ABB RAPID module: Module1.mod

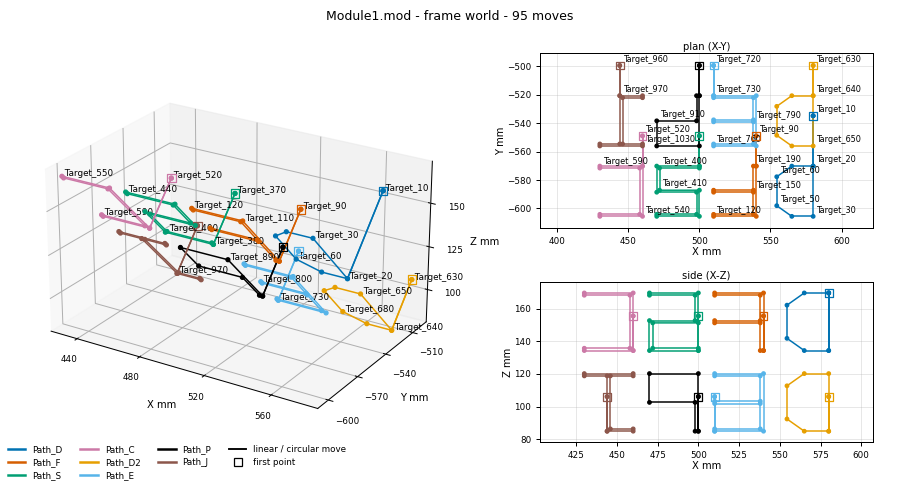
[picture p0: tool path of Module1.mod in frame world, 95 of 99 moves have a stored position in this frame; points joined in program order, loops and branches not executed]
MODULE Module1




    PERS tooldata PortaMarcadorTCP:=[TRUE,[[0,0,152],[1,0,0,0]],[0.15,[0,0,65],[1,0,0,0],0,0,0]];
    TASK PERS wobjdata Tablero_Inclinado:=[FALSE,TRUE,"",[[600,-619.706,183.848],[0,0,0.923879533,-0.382683432]],[[0,0,0],[1,0,0,0]]];
    CONST robtarget Target_10:=[[20,70,-50],[1,0,0,0],[-1,-1,0,0],[9E+09,9E+09,9E+09,9E+09,9E+09,9E+09]];
    CONST robtarget Target_20:=[[20,70.000430916,-0.000095827],[1,0,0,0],[-1,-1,0,0],[9E+09,9E+09,9E+09,9E+09,9E+09,9E+09]];
    CONST robtarget Target_30:=[[20,20.000430915,-0.00009588],[1,0,0,0],[-1,-1,0,0],[9E+09,9E+09,9E+09,9E+09,9E+09,9E+09]];
    CONST robtarget Target_40:=[[35,20.000430915,-0.00009588],[1,0,0,0],[-1,-1,0,0],[9E+09,9E+09,9E+09,9E+09,9E+09,9E+09]];
    CONST robtarget Target_50:=[[45.606601718,30.607032633,-0.000095869],[1,0.000000001,0,0],[-1,-1,0,0],[9E+09,9E+09,9E+09,9E+09,9E+09,9E+09]];
    CONST robtarget Target_60:=[[45.606601718,59.393829198,-0.000095838],[1,0,0,0],[-1,-1,0,0],[9E+09,9E+09,9E+09,9E+09,9E+09,9E+09]];
    CONST robtarget Target_70:=[[35,70.000430916,-0.000095827],[1,0.000000001,0,0],[-1,-1,0,0],[9E+09,9E+09,9E+09,9E+09,9E+09,9E+09]];
    CONST robtarget Target_80:=[[20,70.000430916,-0.000095827],[1,0,0,0],[0,0,0,0],[9E+09,9E+09,9E+09,9E+09,9E+09,9E+09]];
    CONST robtarget Target_10_2:=[[20,70,-50],[1,0,0,0],[-1,-1,0,0],[9E+09,9E+09,9E+09,9E+09,9E+09,9E+09]];
    CONST robtarget Target_90:=[[60,70.000430947,-30.000095827],[1,0,0,0],[0,0,0,0],[9E+09,9E+09,9E+09,9E+09,9E+09,9E+09]];
    CONST robtarget Target_100:=[[60,70.000430916,-0.000095827],[1,0,0,0],[-1,-1,0,0],[9E+09,9E+09,9E+09,9E+09,9E+09,9E+09]];
    CONST robtarget Target_110:=[[60,20.000430915,-0.00009588],[1,0,0,0],[-1,-1,0,0],[9E+09,9E+09,9E+09,9E+09,9E+09,9E+09]];
    CONST robtarget Target_120:=[[90,20.000430915,-0.00009588],[1,0,0,0],[-1,-2,0,0],[9E+09,9E+09,9E+09,9E+09,9E+09,9E+09]];
    CONST robtarget Target_130:=[[90,22.000430916,-0.000095877],[1,0,0,0],[-1,-2,0,0],[9E+09,9E+09,9E+09,9E+09,9E+09,9E+09]];
    CONST robtarget Target_140:=[[62,22.000430916,-0.000095877],[1,0,0,0],[-1,-1,0,0],[9E+09,9E+09,9E+09,9E+09,9E+09,9E+09]];
    CONST robtarget Target_150:=[[62,44.000430916,-0.000095854],[1,0,0,0],[-1,-1,0,0],[9E+09,9E+09,9E+09,9E+09,9E+09,9E+09]];
    CONST robtarget Target_160:=[[90,44.000430539,-0.000095855],[1,0,0,0],[-1,-2,0,0],[9E+09,9E+09,9E+09,9E+09,9E+09,9E+09]];
    CONST robtarget Target_170:=[[90,46.000430916,-0.000095852],[1,0,0,0],[-1,-2,0,0],[9E+09,9E+09,9E+09,9E+09,9E+09,9E+09]];
    CONST robtarget Target_180:=[[62,46.000430916,-0.000095852],[1,0,0,0],[-1,-1,0,0],[9E+09,9E+09,9E+09,9E+09,9E+09,9E+09]];
    CONST robtarget Target_190:=[[62,70.000430916,-0.000095827],[1,0,0,0],[-1,-2,0,0],[9E+09,9E+09,9E+09,9E+09,9E+09,9E+09]];
    CONST robtarget Target_200:=[[60,70.000430916,-0.000095827],[1,0,0,0],[-1,-1,0,0],[9E+09,9E+09,9E+09,9E+09,9E+09,9E+09]];
    CONST robtarget Target_210:=[[60,70.000430947,-30.000095827],[1,0,0,0],[-1,-1,0,0],[9E+09,9E+09,9E+09,9E+09,9E+09,9E+09]];
    CONST robtarget Target_370:=[[100,70.000430703,-30.000095827],[1,0,0,0],[-1,-2,0,0],[9E+09,9E+09,9E+09,9E+09,9E+09,9E+09]];
    CONST robtarget Target_380:=[[100,70.00043067,-0.000095827],[1,0,0,0],[-1,-2,0,0],[9E+09,9E+09,9E+09,9E+09,9E+09,9E+09]];
    CONST robtarget Target_390:=[[100,68.000430671,-0.000095829],[1,0,0,0],[-1,-2,0,0],[9E+09,9E+09,9E+09,9E+09,9E+09,9E+09]];
    CONST robtarget Target_400:=[[128,68.000430671,-0.000095829],[1,0,0,0],[-1,-2,0,0],[9E+09,9E+09,9E+09,9E+09,9E+09,9E+09]];
    CONST robtarget Target_410:=[[127.999999808,46.000430671,-0.000095852],[1,0,0,0],[-1,-2,0,0],[9E+09,9E+09,9E+09,9E+09,9E+09,9E+09]];
    CONST robtarget Target_420:=[[100,45.997147496,-0.000095852],[1,0.000000001,0,0],[-1,-2,0,0],[9E+09,9E+09,9E+09,9E+09,9E+09,9E+09]];
    CONST robtarget Target_430:=[[100,20.000430915,-0.00009588],[1,0,0,0],[-1,-2,0,0],[9E+09,9E+09,9E+09,9E+09,9E+09,9E+09]];
    CONST robtarget Target_440:=[[130,20.000430915,-0.00009588],[1,0,0,0],[-1,-2,0,0],[9E+09,9E+09,9E+09,9E+09,9E+09,9E+09]];
    CONST robtarget Target_450:=[[130,22.000430916,-0.000095877],[1,0,0,0],[-1,-2,0,0],[9E+09,9E+09,9E+09,9E+09,9E+09,9E+09]];
    CONST robtarget Target_460:=[[102,22.000430916,-0.000095877],[1,0,0,0],[-1,-2,0,0],[9E+09,9E+09,9E+09,9E+09,9E+09,9E+09]];
    CONST robtarget Target_470:=[[102,44.000430916,-0.000095854],[1,0,0,0],[-1,-2,0,0],[9E+09,9E+09,9E+09,9E+09,9E+09,9E+09]];
    CONST robtarget Target_480:=[[130,44.00043067,-0.000095855],[1,0,0,0],[-1,-2,0,0],[9E+09,9E+09,9E+09,9E+09,9E+09,9E+09]];
    CONST robtarget Target_490:=[[130,70.00043067,-0.000095827],[1,0,0,0],[-1,-2,0,0],[9E+09,9E+09,9E+09,9E+09,9E+09,9E+09]];
    CONST robtarget Target_500:=[[100,70.00043067,-0.000095827],[1,0,0,0],[-1,-2,0,0],[9E+09,9E+09,9E+09,9E+09,9E+09,9E+09]];
    CONST robtarget Target_510:=[[100,70.000430703,-30.000095827],[1,0,0,0],[-1,-2,0,0],[9E+09,9E+09,9E+09,9E+09,9E+09,9E+09]];
    CONST robtarget Target_520:=[[140,70.000430947,-30.000095827],[1,0,0,0],[-1,-2,0,0],[9E+09,9E+09,9E+09,9E+09,9E+09,9E+09]];
    CONST robtarget Target_530:=[[140,70.000430916,-0.000095827],[1,0,0,0],[-1,-2,0,0],[9E+09,9E+09,9E+09,9E+09,9E+09,9E+09]];
    CONST robtarget Target_540:=[[140,20.000430915,-0.00009588],[1,0,0,0],[-1,-2,0,0],[9E+09,9E+09,9E+09,9E+09,9E+09,9E+09]];
    CONST robtarget Target_550:=[[170,20.000430915,-0.00009588],[1,0,0,0],[-1,-2,0,0],[9E+09,9E+09,9E+09,9E+09,9E+09,9E+09]];
    CONST robtarget Target_560:=[[170,22.000431324,-0.000095877],[1,0,0,0],[-1,-2,0,0],[9E+09,9E+09,9E+09,9E+09,9E+09,9E+09]];
    CONST robtarget Target_570:=[[142,22.000430916,-0.000095877],[1,0,0,0],[-1,-2,0,0],[9E+09,9E+09,9E+09,9E+09,9E+09,9E+09]];
    CONST robtarget Target_580:=[[142,68.000430916,-0.000095829],[1,0,0,0],[-1,-2,0,0],[9E+09,9E+09,9E+09,9E+09,9E+09,9E+09]];
    CONST robtarget Target_590:=[[170,68.000430916,-0.000095829],[1,0,0,0],[-1,-2,0,0],[9E+09,9E+09,9E+09,9E+09,9E+09,9E+09]];
    CONST robtarget Target_600:=[[170,70.000430916,-0.000095827],[1,0,0,0],[-1,-2,0,0],[9E+09,9E+09,9E+09,9E+09,9E+09,9E+09]];
    CONST robtarget Target_610:=[[140,70.000430916,-0.000095827],[1,0,0,0],[-1,-2,0,0],[9E+09,9E+09,9E+09,9E+09,9E+09,9E+09]];
    CONST robtarget Target_620:=[[140,70.000430947,-30.000095827],[1,0,0,0],[-1,-2,0,0],[9E+09,9E+09,9E+09,9E+09,9E+09,9E+09]];
    CONST jointtarget PosicionInicial:=[[0,0,0,0,0,0],[9E+09,9E+09,9E+09,9E+09,9E+09,9E+09]];
    CONST jointtarget Intermedio:=[[0,30,0,0,0,0],[9E+09,9E+09,9E+09,9E+09,9E+09,9E+09]];
    CONST robtarget Target_630:=[[20,140.000430947,-30.000095754],[1,0,0,0],[0,0,0,0],[9E+09,9E+09,9E+09,9E+09,9E+09,9E+09]];
    CONST robtarget Target_640:=[[20,140.000430916,-0.000095753],[1,0,0,0],[0,0,0,0],[9E+09,9E+09,9E+09,9E+09,9E+09,9E+09]];
    CONST robtarget Target_650:=[[20,90.000430915,-0.000095806],[1,0,0,0],[0,0,0,0],[9E+09,9E+09,9E+09,9E+09,9E+09,9E+09]];
    CONST robtarget Target_660:=[[35,90.000430915,-0.000095806],[1,0,0,0],[0,0,0,0],[9E+09,9E+09,9E+09,9E+09,9E+09,9E+09]];
    CONST robtarget Target_670:=[[45.606601718,100.607032633,-0.000095795],[1,0.000000001,0,0],[0,0,0,0],[9E+09,9E+09,9E+09,9E+09,9E+09,9E+09]];
    CONST robtarget Target_680:=[[45.606601718,129.393829198,-0.000095764],[1,0,0,0],[0,0,0,0],[9E+09,9E+09,9E+09,9E+09,9E+09,9E+09]];
    CONST robtarget Target_690:=[[35,140.000430916,-0.000095753],[1,0.000000001,0,0],[0,0,0,0],[9E+09,9E+09,9E+09,9E+09,9E+09,9E+09]];
    CONST robtarget Target_700:=[[20,140.000430916,-0.000095753],[1,0,0,0],[0,0,0,0],[9E+09,9E+09,9E+09,9E+09,9E+09,9E+09]];
    CONST robtarget Target_710:=[[20,140.000430947,-30.000095754],[1,0,0,0],[0,0,0,0],[9E+09,9E+09,9E+09,9E+09,9E+09,9E+09]];
    CONST robtarget Target_720:=[[90,140.000430947,-30.000095754],[1,0,0,0],[0,0,0,0],[9E+09,9E+09,9E+09,9E+09,9E+09,9E+09]];
    CONST robtarget Target_730:=[[90,140.000430916,-0.000095753],[1,0,0,0],[0,0,0,0],[9E+09,9E+09,9E+09,9E+09,9E+09,9E+09]];
    CONST robtarget Target_740:=[[60,140.000430916,-0.000095753],[1,0,0,0],[0,0,0,0],[9E+09,9E+09,9E+09,9E+09,9E+09,9E+09]];
    CONST robtarget Target_750:=[[60,90.000430915,-0.000095806],[1,0,0,0],[0,0,0,0],[9E+09,9E+09,9E+09,9E+09,9E+09,9E+09]];
    CONST robtarget Target_760:=[[90,90.000430915,-0.000095806],[1,0,0,0],[0,0,0,0],[9E+09,9E+09,9E+09,9E+09,9E+09,9E+09]];
    CONST robtarget Target_770:=[[90,92.000430916,-0.000095803],[1,0,0,0],[0,0,0,0],[9E+09,9E+09,9E+09,9E+09,9E+09,9E+09]];
    CONST robtarget Target_780:=[[62,92.000430916,-0.000095803],[1,0,0,0],[0,0,0,0],[9E+09,9E+09,9E+09,9E+09,9E+09,9E+09]];
    CONST robtarget Target_790:=[[62,114.000430915,-0.00009578],[1,0,0,0],[0,0,0,0],[9E+09,9E+09,9E+09,9E+09,9E+09,9E+09]];
    CONST robtarget Target_800:=[[90,114.000430592,-0.00009578],[1,0,0,0],[0,0,0,0],[9E+09,9E+09,9E+09,9E+09,9E+09,9E+09]];
    CONST robtarget Target_810:=[[90,116.000430916,-0.000095779],[1,0,0,0],[0,0,0,0],[9E+09,9E+09,9E+09,9E+09,9E+09,9E+09]];
    CONST robtarget Target_820:=[[62,116.000430916,-0.000095779],[1,0,0,0],[0,0,0,0],[9E+09,9E+09,9E+09,9E+09,9E+09,9E+09]];
    CONST robtarget Target_830:=[[62,138.000430915,-0.000095756],[1,0,0,0],[0,0,0,0],[9E+09,9E+09,9E+09,9E+09,9E+09,9E+09]];
    CONST robtarget Target_840:=[[90,138.000430915,-0.000095756],[1,0,0,0],[0,0,0,0],[9E+09,9E+09,9E+09,9E+09,9E+09,9E+09]];
    CONST robtarget Target_850:=[[90,140.000430916,-0.000095753],[1,0,0,0],[0,0,0,0],[9E+09,9E+09,9E+09,9E+09,9E+09,9E+09]];
    CONST robtarget Target_860:=[[90,140.000430947,-30.000095754],[1,0,0,0],[0,0,0,0],[9E+09,9E+09,9E+09,9E+09,9E+09,9E+09]];
    CONST robtarget Target_870:=[[100,140.000430947,-30.000095754],[1,0,0,0],[0,0,0,0],[9E+09,9E+09,9E+09,9E+09,9E+09,9E+09]];
    CONST robtarget Target_880:=[[100,140.000430916,-0.000095753],[1,0,0,0],[0,0,0,0],[9E+09,9E+09,9E+09,9E+09,9E+09,9E+09]];
    CONST robtarget Target_890:=[[100,90.000430915,-0.000095806],[1,0,0,0],[0,0,0,0],[9E+09,9E+09,9E+09,9E+09,9E+09,9E+09]];
    CONST robtarget Target_900:=[[130,90.000430915,-0.000095806],[1,0,0,0],[0,0,0,0],[9E+09,9E+09,9E+09,9E+09,9E+09,9E+09]];
    CONST robtarget Target_910:=[[130,115.000430916,-0.00009578],[1,0,0,0],[0,0,0,0],[9E+09,9E+09,9E+09,9E+09,9E+09,9E+09]];
    CONST robtarget Target_920:=[[102,115.000430916,-0.00009578],[1,0,0,0],[0,0,0,0],[9E+09,9E+09,9E+09,9E+09,9E+09,9E+09]];
    CONST robtarget Target_930:=[[102,140.000430916,-0.000095753],[1,0,0,0],[0,0,0,0],[9E+09,9E+09,9E+09,9E+09,9E+09,9E+09]];
    CONST robtarget Target_940:=[[100,140.000430916,-0.000095753],[1,0,0,0],[0,0,0,0],[9E+09,9E+09,9E+09,9E+09,9E+09,9E+09]];
    CONST robtarget Target_950:=[[100,140.000430947,-30.000095754],[1,0,0,0],[0,0,0,0],[9E+09,9E+09,9E+09,9E+09,9E+09,9E+09]];
    CONST robtarget Target_960:=[[156,140.000430947,-30.000095754],[1,0,0,0],[0,0,0,0],[9E+09,9E+09,9E+09,9E+09,9E+09,9E+09]];
    CONST robtarget Target_970:=[[156,140.000430916,-0.000095753],[1,0,0,0],[0,0,0,0],[9E+09,9E+09,9E+09,9E+09,9E+09,9E+09]];
    CONST robtarget Target_980:=[[140,140.000430916,-0.000095753],[1,0,0,0],[0,0,0,0],[9E+09,9E+09,9E+09,9E+09,9E+09,9E+09]];
    CONST robtarget Target_990:=[[140,138.000430915,-0.000095756],[1,0,0,0],[0,0,0,0],[9E+09,9E+09,9E+09,9E+09,9E+09,9E+09]];
    CONST robtarget Target_1000:=[[154,138.000430915,-0.000095756],[1,0,0,0],[0,0,0,0],[9E+09,9E+09,9E+09,9E+09,9E+09,9E+09]];
    CONST robtarget Target_1010:=[[154,92.000430916,-0.000095803],[1,0,0,0],[0,0,0,0],[9E+09,9E+09,9E+09,9E+09,9E+09,9E+09]];
    CONST robtarget Target_1020:=[[140,92.00043112,-0.000095804],[1,0,0,0],[0,0,0,0],[9E+09,9E+09,9E+09,9E+09,9E+09,9E+09]];
    CONST robtarget Target_1030:=[[140,90.000430915,-0.000095806],[1,0,0,0],[0,0,0,0],[9E+09,9E+09,9E+09,9E+09,9E+09,9E+09]];
    CONST robtarget Target_1040:=[[170,90.000430915,-0.000095806],[1,0,0,0],[0,0,0,0],[9E+09,9E+09,9E+09,9E+09,9E+09,9E+09]];
    CONST robtarget Target_1050:=[[170,92.000430916,-0.000095803],[1,0,0,0],[0,0,0,0],[9E+09,9E+09,9E+09,9E+09,9E+09,9E+09]];
    CONST robtarget Target_1060:=[[156,92.000430916,-0.000095803],[1,0,0,0],[0,0,0,0],[9E+09,9E+09,9E+09,9E+09,9E+09,9E+09]];
    CONST robtarget Target_1070:=[[156,140.000430916,-0.000095753],[1,0,0,0],[0,0,0,0],[9E+09,9E+09,9E+09,9E+09,9E+09,9E+09]];
    CONST robtarget Target_1080:=[[156,140.000430947,-30.000095754],[1,0,0,0],[0,0,0,0],[9E+09,9E+09,9E+09,9E+09,9E+09,9E+09]];
    CONST jointtarget Cambiar_Tool:=[[90,30,-30,0,0,0],[9E+09,9E+09,9E+09,9E+09,9E+09,9E+09]];
    CONST jointtarget Cambiar_Tool_Intermedio:=[[0,0,-90,0,0,0],[9E+09,9E+09,9E+09,9E+09,9E+09,9E+09]];
    VAR num Contador:=0;
    VAR bool off:= FALSE;

    PROC main()
        PosInicial;
        SetDO DO_04,0;
        IF DI_01=1 THEN
            SetDO DO_04,1;
            Acercamiento;
            Path_D;
            Path_F;
            Path_S;
            Path_C;
            Path_D;
            Path_E;
            Path_P;
            Path_J;
            PosInicial;
            SetDO DO_04,0;
        ELSEIF DI_02=1 THEN
            SetDO DO_05,1;
            Mantenimiento_Acercamiento;
            Mantenimiento;
            SetDO DO_05,0;
            WaitUntil DI_01=1 AND DI_02=1;
            SetDO DO_05,1;
            WaitUntil DI_01=0 AND DI_02=0;
            SetDO DO_05,0;
            WaitUntil DI_01=1 AND DI_02=1;
            SetDO DO_05,1;
            WaitUntil DI_01=0 AND DI_02=0;
            Mantenimiento_Acercamiento;
            PosInicial;
            SetDO DO_05,0;
        ENDIF
    ENDPROC

    PROC Apagar()
        IF off = FALSE THEN
            IF Contador<3 AND DI_01=1 AND DI_02=1 THEN
                WaitTime 1;
                Contador:= Contador+1;
                Apagar;
            ELSEIF Contador>=3 THEN
                off:= TRUE;
                Contador:=0;
            ENDIF
        ELSE
            IF Contador<3 AND DI_01=1 AND DI_02=1 THEN
                WaitTime 1;
                Contador:= Contador+1;
                Apagar;
            ELSEIF Contador>=3 THEN
                off:= False;
                Contador:=0;
            ENDIF
            main;
        ENDIF
    ENDPROC

    PROC Path_D()
        MoveJ Target_10,v150,z5,PortaMarcadorTCP\WObj:=Tablero_Inclinado;
        MoveL Target_10,v200,z5,PortaMarcadorTCP\WObj:=Tablero_Inclinado;
        MoveL Target_20,v200,z5,PortaMarcadorTCP\WObj:=Tablero_Inclinado;
        MoveL Target_30,v200,z5,PortaMarcadorTCP\WObj:=Tablero_Inclinado;
        MoveL Target_40,v200,z5,PortaMarcadorTCP\WObj:=Tablero_Inclinado;
        MoveL Target_50,v200,z5,PortaMarcadorTCP\WObj:=Tablero_Inclinado;
        MoveL Target_60,v200,z5,PortaMarcadorTCP\WObj:=Tablero_Inclinado;
        MoveL Target_70,v200,z5,PortaMarcadorTCP\WObj:=Tablero_Inclinado;
        MoveL Target_80,v200,z5,PortaMarcadorTCP\WObj:=Tablero_Inclinado;
        MoveL Target_10_2,v200,z5,PortaMarcadorTCP\WObj:=Tablero_Inclinado;
    ENDPROC
    PROC Path_F()
        MoveL Target_90,v200,z5,PortaMarcadorTCP\WObj:=Tablero_Inclinado;
        MoveL Target_100,v100,z5,PortaMarcadorTCP\WObj:=Tablero_Inclinado;
        MoveL Target_110,v100,z1,PortaMarcadorTCP\WObj:=Tablero_Inclinado;
        MoveL Target_120,v100,z1,PortaMarcadorTCP\WObj:=Tablero_Inclinado;
        MoveL Target_130,v100,z1,PortaMarcadorTCP\WObj:=Tablero_Inclinado;
        MoveL Target_140,v100,z5,PortaMarcadorTCP\WObj:=Tablero_Inclinado;
        MoveL Target_150,v100,z5,PortaMarcadorTCP\WObj:=Tablero_Inclinado;
        MoveL Target_160,v100,z5,PortaMarcadorTCP\WObj:=Tablero_Inclinado;
        MoveL Target_170,v100,z5,PortaMarcadorTCP\WObj:=Tablero_Inclinado;
        MoveL Target_180,v100,z5,PortaMarcadorTCP\WObj:=Tablero_Inclinado;
        MoveL Target_190,v100,z5,PortaMarcadorTCP\WObj:=Tablero_Inclinado;
        MoveL Target_200,v100,z5,PortaMarcadorTCP\WObj:=Tablero_Inclinado;
        MoveL Target_210,v100,z5,PortaMarcadorTCP\WObj:=Tablero_Inclinado;
    ENDPROC
    PROC Path_S()
        MoveL Target_370,v100,z1,PortaMarcadorTCP\WObj:=Tablero_Inclinado;
        MoveL Target_380,v100,z1,PortaMarcadorTCP\WObj:=Tablero_Inclinado;
        MoveL Target_390,v100,z1,PortaMarcadorTCP\WObj:=Tablero_Inclinado;
        MoveL Target_400,v100,z1,PortaMarcadorTCP\WObj:=Tablero_Inclinado;
        MoveL Target_410,v100,z1,PortaMarcadorTCP\WObj:=Tablero_Inclinado;
        MoveL Target_420,v100,z1,PortaMarcadorTCP\WObj:=Tablero_Inclinado;
        MoveL Target_430,v100,z1,PortaMarcadorTCP\WObj:=Tablero_Inclinado;
        MoveL Target_440,v100,z1,PortaMarcadorTCP\WObj:=Tablero_Inclinado;
        MoveL Target_450,v100,z1,PortaMarcadorTCP\WObj:=Tablero_Inclinado;
        MoveL Target_460,v100,z1,PortaMarcadorTCP\WObj:=Tablero_Inclinado;
        MoveL Target_470,v100,z1,PortaMarcadorTCP\WObj:=Tablero_Inclinado;
        MoveL Target_480,v100,z1,PortaMarcadorTCP\WObj:=Tablero_Inclinado;
        MoveL Target_490,v100,z1,PortaMarcadorTCP\WObj:=Tablero_Inclinado;
        MoveL Target_500,v100,z1,PortaMarcadorTCP\WObj:=Tablero_Inclinado;
        MoveL Target_510,v100,z1,PortaMarcadorTCP\WObj:=Tablero_Inclinado;
    ENDPROC
    PROC Path_C()
        MoveL Target_520,v100,z1,PortaMarcadorTCP\WObj:=Tablero_Inclinado;
        MoveL Target_530,v100,z1,PortaMarcadorTCP\WObj:=Tablero_Inclinado;
        MoveL Target_540,v100,z1,PortaMarcadorTCP\WObj:=Tablero_Inclinado;
        MoveL Target_550,v100,z1,PortaMarcadorTCP\WObj:=Tablero_Inclinado;
        MoveL Target_560,v100,z1,PortaMarcadorTCP\WObj:=Tablero_Inclinado;
        MoveL Target_570,v100,z1,PortaMarcadorTCP\WObj:=Tablero_Inclinado;
        MoveL Target_580,v100,z1,PortaMarcadorTCP\WObj:=Tablero_Inclinado;
        MoveL Target_590,v100,z1,PortaMarcadorTCP\WObj:=Tablero_Inclinado;
        MoveL Target_600,v100,z1,PortaMarcadorTCP\WObj:=Tablero_Inclinado;
        MoveL Target_610,v100,z1,PortaMarcadorTCP\WObj:=Tablero_Inclinado;
        MoveL Target_620,v100,z1,PortaMarcadorTCP\WObj:=Tablero_Inclinado;
    ENDPROC
    PROC PosInicial()
        MoveAbsJ PosicionInicial,v200,z100,PortaMarcadorTCP\WObj:=Tablero_Inclinado;
    ENDPROC
    PROC Acercamiento()
        MoveAbsJ Intermedio,v150,z100,PortaMarcadorTCP\WObj:=Tablero_Inclinado;
    ENDPROC
    PROC Path_D2()
        MoveL Target_630,v200,z1,PortaMarcadorTCP\WObj:=Tablero_Inclinado;
        MoveL Target_640,v200,z1,PortaMarcadorTCP\WObj:=Tablero_Inclinado;
        MoveL Target_650,v200,z1,PortaMarcadorTCP\WObj:=Tablero_Inclinado;
        MoveL Target_660,v200,z1,PortaMarcadorTCP\WObj:=Tablero_Inclinado;
        MoveL Target_670,v200,z1,PortaMarcadorTCP\WObj:=Tablero_Inclinado;
        MoveL Target_680,v200,z1,PortaMarcadorTCP\WObj:=Tablero_Inclinado;
        MoveL Target_690,v200,z1,PortaMarcadorTCP\WObj:=Tablero_Inclinado;
        MoveL Target_700,v200,z1,PortaMarcadorTCP\WObj:=Tablero_Inclinado;
        MoveL Target_710,v200,z1,PortaMarcadorTCP\WObj:=Tablero_Inclinado;
    ENDPROC
    PROC Path_E()
        MoveL Target_720,v100,z1,PortaMarcadorTCP\WObj:=Tablero_Inclinado;
        MoveL Target_730,v100,z1,PortaMarcadorTCP\WObj:=Tablero_Inclinado;
        MoveL Target_740,v100,z1,PortaMarcadorTCP\WObj:=Tablero_Inclinado;
        MoveL Target_750,v100,z1,PortaMarcadorTCP\WObj:=Tablero_Inclinado;
        MoveL Target_760,v100,z1,PortaMarcadorTCP\WObj:=Tablero_Inclinado;
        MoveL Target_770,v100,z1,PortaMarcadorTCP\WObj:=Tablero_Inclinado;
        MoveL Target_780,v100,z1,PortaMarcadorTCP\WObj:=Tablero_Inclinado;
        MoveL Target_790,v100,z1,PortaMarcadorTCP\WObj:=Tablero_Inclinado;
        MoveL Target_800,v100,z1,PortaMarcadorTCP\WObj:=Tablero_Inclinado;
        MoveL Target_810,v100,z1,PortaMarcadorTCP\WObj:=Tablero_Inclinado;
        MoveL Target_820,v100,z1,PortaMarcadorTCP\WObj:=Tablero_Inclinado;
        MoveL Target_830,v100,z1,PortaMarcadorTCP\WObj:=Tablero_Inclinado;
        MoveL Target_840,v100,z1,PortaMarcadorTCP\WObj:=Tablero_Inclinado;
        MoveL Target_850,v100,z1,PortaMarcadorTCP\WObj:=Tablero_Inclinado;
        MoveL Target_860,v100,z1,PortaMarcadorTCP\WObj:=Tablero_Inclinado;
    ENDPROC
    PROC Path_P()
        MoveL Target_870,v150,z1,PortaMarcadorTCP\WObj:=Tablero_Inclinado;
        MoveL Target_880,v150,z1,PortaMarcadorTCP\WObj:=Tablero_Inclinado;
        MoveL Target_890,v150,z1,PortaMarcadorTCP\WObj:=Tablero_Inclinado;
        MoveL Target_900,v150,z1,PortaMarcadorTCP\WObj:=Tablero_Inclinado;
        MoveL Target_910,v150,z1,PortaMarcadorTCP\WObj:=Tablero_Inclinado;
        MoveL Target_920,v150,z1,PortaMarcadorTCP\WObj:=Tablero_Inclinado;
        MoveL Target_930,v150,z1,PortaMarcadorTCP\WObj:=Tablero_Inclinado;
        MoveL Target_940,v150,z1,PortaMarcadorTCP\WObj:=Tablero_Inclinado;
        MoveL Target_950,v150,z1,PortaMarcadorTCP\WObj:=Tablero_Inclinado;
    ENDPROC
    PROC Path_J()
        MoveL Target_960,v150,z1,PortaMarcadorTCP\WObj:=Tablero_Inclinado;
        MoveL Target_970,v150,z1,PortaMarcadorTCP\WObj:=Tablero_Inclinado;
        MoveL Target_980,v150,z1,PortaMarcadorTCP\WObj:=Tablero_Inclinado;
        MoveL Target_990,v150,z1,PortaMarcadorTCP\WObj:=Tablero_Inclinado;
        MoveL Target_1000,v150,z1,PortaMarcadorTCP\WObj:=Tablero_Inclinado;
        MoveL Target_1010,v150,z1,PortaMarcadorTCP\WObj:=Tablero_Inclinado;
        MoveL Target_1020,v150,z1,PortaMarcadorTCP\WObj:=Tablero_Inclinado;
        MoveL Target_1030,v150,z1,PortaMarcadorTCP\WObj:=Tablero_Inclinado;
        MoveL Target_1040,v150,z1,PortaMarcadorTCP\WObj:=Tablero_Inclinado;
        MoveL Target_1050,v150,z1,PortaMarcadorTCP\WObj:=Tablero_Inclinado;
        MoveL Target_1060,v150,z1,PortaMarcadorTCP\WObj:=Tablero_Inclinado;
        MoveL Target_1070,v150,z1,PortaMarcadorTCP\WObj:=Tablero_Inclinado;
        MoveL Target_1080,v150,z1,PortaMarcadorTCP\WObj:=Tablero_Inclinado;
    ENDPROC
    PROC Mantenimiento()
        MoveAbsJ Cambiar_Tool,v100,z100,PortaMarcadorTCP\WObj:=Tablero_Inclinado;
    ENDPROC
    PROC Mantenimiento_Acercamiento()
        MoveAbsJ Cambiar_Tool_Intermedio,v100,z100,PortaMarcadorTCP\WObj:=Tablero_Inclinado;
    ENDPROC
ENDMODULE
